INTERFACE itfSynchronizedAxisCommand EXTENDS itfAxisCommand

PROPERTY InSync : BOOL
GET
END_GET
END_PROPERTY

END_INTERFACE

(* stored: Version 1.1.0.1, ProductVersion 3.1.4024.12
   Itf itfSynchronizedAxisCommand: Id {57e46a7a-22f5-473d-bd21-af003d437965}
   Property InSync: Id {4c6be8ac-11ee-419f-807f-8d4fb4150cce}
   Get Get: Id {3e770395-ebea-4f4f-a010-b4bade2560b7} *)
